(* PLC project Generated.project, CODESYS CODESYS V3.5 SP19 Patch 1 *)
(* stored: creationDateTime 2026-08-28T11:10:17.718047, modificationDateTime 2026-08-28T11:10:17.718047 *)

(* values of E_ProgramSequence: NONE: Aucune séquence active; MAIN_CYCLE: Cycle principal automatique de dragage X0..X13; DIVE_SEARCH: Sous-séquence de plongée / recherche de fond; EXTRACTION: Sous-séquence d'extraction et fermeture *)

{attribute 'qualified_only'}
{attribute 'strict'}
TYPE E_ProgramSequence : (NONE := 0, MAIN_CYCLE := 1, DIVE_SEARCH := 2, EXTRACTION := 3);
END_TYPE
